{attribute 'linkalways'} 
{attribute 'no_explicit_call' := 'This FB is a CLASS and must be accessed using methods or properties'}
{attribute 'enable_dynamic_creation'}
FUNCTION_BLOCK Node_F_VN_FillContainer_DINT EXTENDS VisionNode
VAR
    ipContainer : _ITcVnContainer;
    nValue : _DINT(0);
    hrPrev : _HRESULT(S_OK);
    hresult : _HRESULT(S_OK);
END_VAR

METHOD PUBLIC  Clone : I_Node
VAR
    pNode : POINTER TO Node_F_VN_FillContainer_DINT;
END_VAR
pNode := __NEW(Node_F_VN_FillContainer_DINT);
Clone := pNode^;
END_METHOD

METHOD FB_init : BOOL
VAR_INPUT
    bInitRetains : BOOL; // if TRUE, the retain variables are initialized (warm start / cold start)
    bInCopyCode : BOOL;  // if TRUE, the instance afterwards gets moved into the copy code (online change)
END_VAR
AddInput('ipContainer', ipContainer);
AddInput('nValue', nValue);
AddInput('hrPrev', hrPrev);
AddOutput('ipContainer', ipContainer);
AddOutput('hresult',hresult);
END_METHOD

METHOD PROTECTED OnExecute : HRESULT
hresult.Value := F_VN_FillContainer_DINT(
    ipContainer := ipContainer.Value,
    nValue := nValue.Value,
    hrPrev:= hrPrev.Value);
END_METHOD

METHOD PUBLIC PreExecutionCheck
VAR_INPUT
    Check : I_PreExecutionChecks;
END_VAR
Check.IsTrue(ipContainer.IsValid, 'ipContainer must be a valid container');
END_METHOD

END_FUNCTION_BLOCK

(* stored: Version 1.1.0.1, ProductVersion 3.1.4024.13
   POU Node_F_VN_FillContainer_DINT: Id {88b248b0-a51c-4bf9-95f3-58458d79c61c}, SpecialFunc None
   Folder Constructor: Id {6c57ef5a-fb99-445b-873b-06c354fe3ca3}
   Method Clone: Id {b27a2c68-a24c-4f77-99ee-310d121fec9b}
   Method FB_init: Id {24987666-6b65-4ee2-aa8d-984cc861a7e1}
   Method OnExecute: Id {022f44cd-411d-4ff7-b73e-a2a56f1a9260}
   Method PreExecutionCheck: Id {67db0e9e-aa86-4457-849f-6a0b96e51225} *)
